// List of Strings.
FUNCTION_BLOCK FB_TargList
VAR
	List : ARRAY[ 0 .. GVL_List.LIST_SIZE - 1 ] OF T_Arg; // hold list
	_Count : UDINT := 0; // number of items.
END_VAR

// Add item to list. TRUE if successful. 
METHOD PUBLIC AddItem : BOOL
VAR_INPUT
	Item : T_Arg; // item to add.
END_VAR
IF _Count < GVL_List.LIST_SIZE THEN
	List[_Count] := Item; // list is zero indexed, so number of items points at next free space.
	_Count := _Count + 1; 
	AddItem := TRUE;
END_IF
END_METHOD

// Removes all list items
METHOD PUBLIC Clear
MEMSET(ADR(List[0]), 0, SIZEOF(List));
_Count := 0;
END_METHOD

// TRUE if Item is in FB_List.
METHOD PUBLIC Contains : BOOL
VAR_INPUT
	Item : T_Arg; // Item to check.
END_VAR
Contains := FindIndex(Item) >= 0;
END_METHOD

{attribute 'monitoring' := 'call'}
// Number of items in list.
PROPERTY PUBLIC Count : UDINT
GET
Count := _Count;
END_GET
END_PROPERTY

METHOD PUBLIC FindIndex : INT
VAR_INPUT
	Item : T_Arg; // Item to check.
END_VAR
VAR
	i : UINT := 0;
END_VAR
FindIndex := -1;
i := 0;
WHILE ( (FindIndex < 0) AND (i < _Count) ) DO
	
	FindIndex := SEL(Item = List[i], FindIndex, TO_INT(i) ); // if it matches, return the position.
	i := i + 1;
	
END_WHILE
END_METHOD

// Return item in list at index position. Returns empty string if invalid index.
METHOD PUBLIC GetIndex : T_Arg
VAR_INPUT
	Index : UDINT;
END_VAR
THIS^.TryGetIndex(Index,  GetIndex);
END_METHOD

//Remove the specified index. Shuffle remaining so list is intact.
METHOD PUBLIC RemoveIndex : BOOL
VAR_INPUT
	Index : UDINT;
END_VAR
IF Index >= _Count THEN // invalid index request.
	RETURN;
END_IF

IF Index < _Count - 1 THEN // If Index = _Count -1, last two lines sufficient.

	MEMMOVE( 
		destAddr := ADR( List[Index] ), 
		srcAddr := ADR( List[Index + 1] ), 
		n := SIZEOF(List[0]) * (_Count - Index - 1)
	);
	
END_IF

RemoveIndex := TRUE;
MEMSET(ADR(List[_Count - 1]), 0, SIZEOF(T_Arg));
_Count := _Count - 1; // reduce count.
END_METHOD

// TRUE if successful and list item in sItem
METHOD PUBLIC TryGetIndex : BOOL
VAR_INPUT
	Index : UDINT;
END_VAR
VAR_IN_OUT
	Item : T_Arg;
END_VAR
IF Index < _Count THEN
	TryGetIndex := TRUE;
	Item := List[Index];
END_IF
END_METHOD

END_FUNCTION_BLOCK

(* stored: Version 1.1.0.1, ProductVersion 3.1.4020.12
   POU FB_TargList: Id {618d746f-d289-47af-ba3d-b2ba9dc07772}, SpecialFunc None
   Method AddItem: Id {9e016b54-56df-4e2b-85b0-f604d5c30bc0}
   Method Clear: Id {8f768700-0070-4763-b654-ecdb9354e2b8}
   Method Contains: Id {924f2197-aee4-4a0e-a924-ceba24bd6410}
   Property Count: Id {ea805cf5-f90e-4089-a198-e5f95d09b44b}
   Get Get: Id {d9137fce-ae3e-4123-bd30-4446a91b9690}
   Method FindIndex: Id {a804a17e-940b-4212-abfe-c9f67ce123f8}
   Method GetIndex: Id {62e1a232-c66b-48da-8ffe-c2567273ec59}
   Method RemoveIndex: Id {8615e590-49d3-42f1-be26-373da1e4c532}
   Method TryGetIndex: Id {1131e0e2-5709-420c-ad2b-868ce8b81f75} *)
